FUNCTION_BLOCK FB_NaiveFF
VAR_INPUT
	fPs 		: LREAL; // [bar]
	fPa 		: LREAL; // [bar]
	fPb 		: LREAL; // [bar]
	
	fXDotRef 	: LREAL; // [m/s]
END_VAR
VAR_OUTPUT

	fFF 		: LREAL; // [-1..1], Spool signal for position, u
	fFlow 		: LREAL; // [l/min]
	fKv 		: LREAL; // [l/min / bar^0.5]
END_VAR
VAR
	fDeltaP		: LREAL; // [bar]
END_VAR




IF fXDotRef > 0.0 THEN
	fFlow := fXDotRef * G_Parameter.fAreaUp * 6E4;
	fDeltaP := fPs - fPa;
	
	fFF := -(0.2143 + 0.7857 * fKv/3.7796);
ELSIF fXDotRef < 0.0 THEN
	fFlow := fXDotRef * G_Parameter.fAreaDown * 6E4;
	fDeltaP := fPs - fPb;
	
	fFF := (0.2143 + 0.7857 * fKv/3.7796);
ELSE
	fFlow := 0.0;
	fFF := 0.0;
END_IF

IF fDeltaP <= 0.0 THEN
	fKv := 4.0;
ELSE
	fKv := ABS(fFlow)/SQRT(fDeltaP);
END_IF

END_FUNCTION_BLOCK

(* stored: Version 1.1.0.1, ProductVersion 3.1.4024.12
   POU FB_NaiveFF: Id {ca7bc146-de72-40c0-8b17-2acf5555ebf6}, SpecialFunc None *)
